// TIA Portal V20 export
// export: Created 2026-07-10T11:12:33.5328435Z, ExportSetting WithDefaults, DisplayName Totally Integrated Automation Portal, DisplayVersion V20, DisplayName TIA Portal Openness, DisplayVersion V20, DisplayName TIA Portal Version Control Interface, DisplayVersion V20, DisplayName STEP 7 Professional, DisplayVersion V20, DisplayName STEP 7 Safety, DisplayVersion V20, DisplayName WinCC Basic/Comfort/Advanced, DisplayVersion V20, DisplayName WinCC Unified, DisplayVersion V20
FUNCTION_BLOCK "MotorMoverToSwitch"   // FB13, SCL
{ S7_Optimized_Access := 'TRUE' }
VERSION : 0.1
// stored: AutoNumber true, IsIECCheckEnabled false, IsRetainMemResEnabled false, MemoryReserve 100, SetENOAutomatically false, UDAEnableTagReadback false
   VAR_INPUT
      Enable : Bool;
      Go : Bool;
      TargetSwitch100 : Bool := True;
      MovePause : Time := T#10s;
      isMoving : Bool;
      LimitSwitch0 : Bool;
      LimitSwitch100 : Bool;
   END_VAR
   VAR_OUTPUT
      Open : Bool;
      Close : Bool;
   END_VAR
   VAR
      GoTo0 : Bool;
      GoTo100 : Bool;
      MovingTOF { S7_SetPoint := 'True'} : TOF_TIME;
   END_VAR
BEGIN
   #MovingTOF(IN:=#isMoving,
              PT:=#MovePause);

   IF #Enable THEN
       IF (NOT #MovingTOF.Q) AND #TargetSwitch100 AND #Go THEN
           #GoTo100 := TRUE;
       END_IF;
       IF #LimitSwitch100 OR (NOT #TargetSwitch100) OR (NOT #Go) THEN
           #GoTo100 := FALSE;
       END_IF;

       IF (NOT #MovingTOF.Q) AND (NOT #TargetSwitch100) AND #Go THEN
           #GoTo0 := #Go;
       END_IF;
       IF #LimitSwitch0 OR #TargetSwitch100 OR (NOT #Go) THEN
           #GoTo0 := FALSE;
       END_IF;

       IF #GoTo100 THEN
           #Open := TRUE;
           #Close := FALSE;
       ELSIF #GoTo0 THEN
           #Open := FALSE;
           #Close := TRUE;
       ELSE
           #Open := FALSE;
           #Close := FALSE;
       END_IF;
   ELSE
       #Open := FALSE;
       #Close := FALSE;
       #GoTo0 := FALSE;
       #GoTo100 := FALSE;
   END_IF;
END_FUNCTION_BLOCK
